PROGRAM MormingBreakfastTask
VAR
	//Variables booleans
	bHungry 			: BOOL;
	bStartPreparation 	: BOOL;
	bStartEat 			: BOOL;
	bReady 				: BOOL;
	//Variables timers
	fbGoToKitchen 		: TON;
	fbDecideIfIEat 		: TON;
	fbPrepareTea 		: TON;
	fbPrepareEggs 		: TON;
	fbPrepareBread 		: TON;
	fbImEating 			: TON;
END_VAR

//First step: Get up and decide if want to eat breakfast

fbDecideIfIEat(IN:=GVL.bGetUp,PT:=T#3S);

IF fbDecideIfIEat.Q THEN
	bHungry := TRUE;
END_IF
fbGoToKitchen(IN:=bHungry,PT:=T#3S);

//Second Step: Now in the kitchen im going to prepare my breakfast

IF fbGoToKitchen.Q THEN
	bStartPreparation := TRUE;
END_IF

fbPrepareTea(IN:=bStartPreparation,PT:=T#7S);     //Im going to use this .Q because it is the last to finish when i cook
fbPrepareBread(IN:=bStartPreparation,PT:=T#3S);
fbPrepareEggs(IN:=bStartPreparation,PT:=T#5S);

//Third step: Finally i end the preparation and start to eat

IF fbPrepareTea.Q AND NOT bStartEat THEN
    bStartEat := TRUE;
END_IF

fbImEating(IN := bStartEat, PT := T#10S);

GVL.bReady := fbImEating.Q;

END_PROGRAM

(* stored: Version 1.1.0.1, ProductVersion 3.1.4024.12
   POU MormingBreakfastTask: Id {b26e7558-b806-4d64-b9a0-6213d32beadb}, SpecialFunc None *)
